// Tests for the command dispatch of BROTLib.FB_Comm_MQTT_Influx (BROTLib#39): single-field messages as pyBROT and
// BROTgui send them, and multi-field messages where track/slew must see the data of the same message. The handler is
// called directly with a payload; no MQTT connection is made. A stub records what it asks the telescope to do.
FUNCTION_BLOCK FB_Comm_MQTT_Influx_Tests EXTENDS TcUnit.FB_TestSuite
VAR
	fbComm	: BROTLib.FB_Comm_MQTT_Influx;
	stub	: FB_TelescopeStub;
	bReady	: BOOL;
	bSingle_Field_Messages_Still_Fill_The_Buffer	: BOOL;
	bData_Before_Verb_In_One_Message	: BOOL;
	bVerb_First_Uses_Data_From_The_Same_Message	: BOOL;
	bSame_Message_Data_Beats_The_Buffer	: BOOL;
	bIncomplete_Pair_Is_Dropped	: BOOL;
	bBuffer_Is_Cleared_After_Track	: BOOL;
	bSlew_Takes_Elevation_And_Azimuth_From_One_Message	: BOOL;
	bTrailing_Timestamp_Does_Not_Break_The_Last_Field	: BOOL;
	bOther_Measurement_Is_Ignored	: BOOL;
	bFields_Beyond_The_Eighth_Are_Ignored	: BOOL;
	bNon_Numeric_Coordinate_Is_Rejected	: BOOL;
	bOut_Of_Range_Coordinates_Are_Rejected	: BOOL;
	bRange_Limits_Are_Accepted	: BOOL;
	bRejected_Value_Clears_The_Buffer	: BOOL;
END_VAR

IF NOT bReady THEN
	bReady := TRUE;
	fbComm.Telescope := stub;
END_IF
Single_Field_Messages_Still_Fill_The_Buffer();
Data_Before_Verb_In_One_Message();
Verb_First_Uses_Data_From_The_Same_Message();
Same_Message_Data_Beats_The_Buffer();
Incomplete_Pair_Is_Dropped();
Buffer_Is_Cleared_After_Track();
Slew_Takes_Elevation_And_Azimuth_From_One_Message();
Trailing_Timestamp_Does_Not_Break_The_Last_Field();
Other_Measurement_Is_Ignored();
Fields_Beyond_The_Eighth_Are_Ignored();
Non_Numeric_Coordinate_Is_Rejected();
Out_Of_Range_Coordinates_Are_Rejected();
Range_Limits_Are_Accepted();
Rejected_Value_Clears_The_Buffer();

// Puts the handler and the stub back to a clean state; every test runs its body once.
METHOD PRIVATE ResetHandler
VAR_INPUT
END_VAR
// drain whatever the previous test left in the handler's buffers: track and slew consume and clear them
fbComm._handleMQTTMessage(sPayloadRcv := 'command track=1');
fbComm._handleMQTTMessage(sPayloadRcv := 'command slew=1');
stub.ClearCounters();
END_METHOD

// The way pyBROT and BROTgui send it today: three messages, the buffer is consumed by track.
METHOD PRIVATE Single_Field_Messages_Still_Fill_The_Buffer
VAR
END_VAR
TEST('Single_Field_Messages_Still_Fill_The_Buffer');
IF NOT bSingle_Field_Messages_Still_Fill_The_Buffer THEN
	bSingle_Field_Messages_Still_Fill_The_Buffer := TRUE;
	ResetHandler();
	fbComm._handleMQTTMessage(sPayloadRcv := 'command rightascension=10.5');
	fbComm._handleMQTTMessage(sPayloadRcv := 'command declination=20.5');
	AssertEquals_INT(Expected := 0, Actual := stub.nTrack, Message := 'before track: number of Track calls');
	fbComm._handleMQTTMessage(sPayloadRcv := 'command track=1');
	AssertEquals_INT(Expected := 1, Actual := stub.nTrack, Message := 'after track: number of Track calls');
	AssertEquals_LREAL(Expected := 10.5, Actual := stub.fTrackRa, Delta := 1.0E-9, Message := 'after track: right ascension');
	AssertEquals_LREAL(Expected := 20.5, Actual := stub.fTrackDec, Delta := 1.0E-9, Message := 'after track: declination');
	TEST_FINISHED();
END_IF
END_METHOD

METHOD PRIVATE Data_Before_Verb_In_One_Message
VAR
END_VAR
TEST('Data_Before_Verb_In_One_Message');
IF NOT bData_Before_Verb_In_One_Message THEN
	bData_Before_Verb_In_One_Message := TRUE;
	ResetHandler();
	fbComm._handleMQTTMessage(sPayloadRcv := 'command rightascension=10.5,declination=20.5,track=1');
	AssertEquals_INT(Expected := 1, Actual := stub.nTrack, Message := 'one message: number of Track calls');
	AssertEquals_LREAL(Expected := 10.5, Actual := stub.fTrackRa, Delta := 1.0E-9, Message := 'one message: right ascension');
	AssertEquals_LREAL(Expected := 20.5, Actual := stub.fTrackDec, Delta := 1.0E-9, Message := 'one message: declination');
	TEST_FINISHED();
END_IF
END_METHOD

// The data pass runs before the verb pass, so the field order does not matter.
METHOD PRIVATE Verb_First_Uses_Data_From_The_Same_Message
VAR
END_VAR
TEST('Verb_First_Uses_Data_From_The_Same_Message');
IF NOT bVerb_First_Uses_Data_From_The_Same_Message THEN
	bVerb_First_Uses_Data_From_The_Same_Message := TRUE;
	ResetHandler();
	fbComm._handleMQTTMessage(sPayloadRcv := 'command track=1,rightascension=10.5,declination=20.5');
	AssertEquals_INT(Expected := 1, Actual := stub.nTrack, Message := 'verb first: number of Track calls');
	AssertEquals_LREAL(Expected := 10.5, Actual := stub.fTrackRa, Delta := 1.0E-9, Message := 'verb first: right ascension');
	AssertEquals_LREAL(Expected := 20.5, Actual := stub.fTrackDec, Delta := 1.0E-9, Message := 'verb first: declination');
	TEST_FINISHED();
END_IF
END_METHOD

// An old buffer value must never be combined with the new target.
METHOD PRIVATE Same_Message_Data_Beats_The_Buffer
VAR
END_VAR
TEST('Same_Message_Data_Beats_The_Buffer');
IF NOT bSame_Message_Data_Beats_The_Buffer THEN
	bSame_Message_Data_Beats_The_Buffer := TRUE;
	ResetHandler();
	fbComm._handleMQTTMessage(sPayloadRcv := 'command rightascension=1.5');
	fbComm._handleMQTTMessage(sPayloadRcv := 'command declination=2.5');
	fbComm._handleMQTTMessage(sPayloadRcv := 'command rightascension=10.5,declination=20.5,track=1');
	AssertEquals_INT(Expected := 1, Actual := stub.nTrack, Message := 'stale buffer: number of Track calls');
	AssertEquals_LREAL(Expected := 10.5, Actual := stub.fTrackRa, Delta := 1.0E-9, Message := 'stale buffer: right ascension');
	AssertEquals_LREAL(Expected := 20.5, Actual := stub.fTrackDec, Delta := 1.0E-9, Message := 'stale buffer: declination');
	TEST_FINISHED();
END_IF
END_METHOD

// Same as the buffered form: no declination, no Track call.
METHOD PRIVATE Incomplete_Pair_Is_Dropped
VAR
END_VAR
TEST('Incomplete_Pair_Is_Dropped');
IF NOT bIncomplete_Pair_Is_Dropped THEN
	bIncomplete_Pair_Is_Dropped := TRUE;
	ResetHandler();
	fbComm._handleMQTTMessage(sPayloadRcv := 'command rightascension=10.5,track=1');
	AssertEquals_INT(Expected := 0, Actual := stub.nTrack, Message := 'declination missing: number of Track calls');
	TEST_FINISHED();
END_IF
END_METHOD

// The second track finds an empty buffer and is dropped, the first call stays the last one.
METHOD PRIVATE Buffer_Is_Cleared_After_Track
VAR
END_VAR
TEST('Buffer_Is_Cleared_After_Track');
IF NOT bBuffer_Is_Cleared_After_Track THEN
	bBuffer_Is_Cleared_After_Track := TRUE;
	ResetHandler();
	fbComm._handleMQTTMessage(sPayloadRcv := 'command rightascension=10.5,declination=20.5,track=1');
	fbComm._handleMQTTMessage(sPayloadRcv := 'command track=1');
	AssertEquals_INT(Expected := 1, Actual := stub.nTrack, Message := 'second track without data: number of Track calls');
	AssertEquals_LREAL(Expected := 10.5, Actual := stub.fTrackRa, Delta := 1.0E-9, Message := 'second track without data: right ascension');
	AssertEquals_LREAL(Expected := 20.5, Actual := stub.fTrackDec, Delta := 1.0E-9, Message := 'second track without data: declination');
	TEST_FINISHED();
END_IF
END_METHOD

METHOD PRIVATE Slew_Takes_Elevation_And_Azimuth_From_One_Message
VAR
END_VAR
TEST('Slew_Takes_Elevation_And_Azimuth_From_One_Message');
IF NOT bSlew_Takes_Elevation_And_Azimuth_From_One_Message THEN
	bSlew_Takes_Elevation_And_Azimuth_From_One_Message := TRUE;
	ResetHandler();
	fbComm._handleMQTTMessage(sPayloadRcv := 'command slew=1,azimuth=120.5,elevation=45.5');
	AssertEquals_INT(Expected := 1, Actual := stub.nSlew, Message := 'slew: number of Slew calls');
	AssertEquals_LREAL(Expected := 120.5, Actual := stub.fSlewAz, Delta := 1.0E-9, Message := 'slew: azimuth');
	AssertEquals_LREAL(Expected := 45.5, Actual := stub.fSlewAlt, Delta := 1.0E-9, Message := 'slew: altitude');
	TEST_FINISHED();
END_IF
END_METHOD

METHOD PRIVATE Trailing_Timestamp_Does_Not_Break_The_Last_Field
VAR
END_VAR
TEST('Trailing_Timestamp_Does_Not_Break_The_Last_Field');
IF NOT bTrailing_Timestamp_Does_Not_Break_The_Last_Field THEN
	bTrailing_Timestamp_Does_Not_Break_The_Last_Field := TRUE;
	ResetHandler();
	fbComm._handleMQTTMessage(sPayloadRcv := 'command rightascension=10.5,declination=20.5,track=1 1700000000000000000');
	AssertEquals_INT(Expected := 1, Actual := stub.nTrack, Message := 'timestamp: number of Track calls');
	AssertEquals_LREAL(Expected := 10.5, Actual := stub.fTrackRa, Delta := 1.0E-9, Message := 'timestamp: right ascension');
	AssertEquals_LREAL(Expected := 20.5, Actual := stub.fTrackDec, Delta := 1.0E-9, Message := 'timestamp: declination');
	TEST_FINISHED();
END_IF
END_METHOD

METHOD PRIVATE Other_Measurement_Is_Ignored
VAR
END_VAR
TEST('Other_Measurement_Is_Ignored');
IF NOT bOther_Measurement_Is_Ignored THEN
	bOther_Measurement_Is_Ignored := TRUE;
	ResetHandler();
	fbComm._handleMQTTMessage(sPayloadRcv := 'status rightascension=10.5,declination=20.5,track=1');
	AssertEquals_INT(Expected := 0, Actual := stub.nTrack, Message := 'measurement status: number of Track calls');
	TEST_FINISHED();
END_IF
END_METHOD

// At most 8 fields per message (a malformed message must not spin the scan cycle); the rest is logged and ignored.
METHOD PRIVATE Fields_Beyond_The_Eighth_Are_Ignored
VAR
END_VAR
TEST('Fields_Beyond_The_Eighth_Are_Ignored');
IF NOT bFields_Beyond_The_Eighth_Are_Ignored THEN
	bFields_Beyond_The_Eighth_Are_Ignored := TRUE;
	ResetHandler();
	fbComm._handleMQTTMessage(sPayloadRcv := 'command rightascension=10.5,declination=20.5,x1=0,x2=0,x3=0,x4=0,x5=0,x6=0,track=1');
	AssertEquals_INT(Expected := 0, Actual := stub.nTrack, Message := 'track is the ninth field: number of Track calls');
	TEST_FINISHED();
END_IF
END_METHOD

// STRING_TO_LREAL turns garbage into 0.0, a valid coordinate; it must not reach Track (#27).
METHOD PRIVATE Non_Numeric_Coordinate_Is_Rejected
VAR
END_VAR
TEST('Non_Numeric_Coordinate_Is_Rejected');
IF NOT bNon_Numeric_Coordinate_Is_Rejected THEN
	bNon_Numeric_Coordinate_Is_Rejected := TRUE;
	ResetHandler();
	fbComm._handleMQTTMessage(sPayloadRcv := 'command rightascension=abc,declination=20.5,track=1');
	AssertEquals_INT(Expected := 0, Actual := stub.nTrack, Message := 'rightascension=abc: number of Track calls');
	fbComm._handleMQTTMessage(sPayloadRcv := 'command rightascension=10.5,declination=nan,track=1');
	AssertEquals_INT(Expected := 0, Actual := stub.nTrack, Message := 'declination=nan: number of Track calls');
	TEST_FINISHED();
END_IF
END_METHOD

METHOD PRIVATE Out_Of_Range_Coordinates_Are_Rejected
VAR
END_VAR
TEST('Out_Of_Range_Coordinates_Are_Rejected');
IF NOT bOut_Of_Range_Coordinates_Are_Rejected THEN
	bOut_Of_Range_Coordinates_Are_Rejected := TRUE;
	ResetHandler();
	fbComm._handleMQTTMessage(sPayloadRcv := 'command rightascension=10.5,declination=95,track=1');
	AssertEquals_INT(Expected := 0, Actual := stub.nTrack, Message := 'declination=95: number of Track calls');
	fbComm._handleMQTTMessage(sPayloadRcv := 'command rightascension=1e999,declination=20.5,track=1');
	AssertEquals_INT(Expected := 0, Actual := stub.nTrack, Message := 'rightascension=1e999: number of Track calls');
	fbComm._handleMQTTMessage(sPayloadRcv := 'command elevation=120,azimuth=10,slew=1');
	AssertEquals_INT(Expected := 0, Actual := stub.nSlew, Message := 'elevation=120: number of Slew calls');
	TEST_FINISHED();
END_IF
END_METHOD

// The limits themselves are valid values; so are signs and exponents.
METHOD PRIVATE Range_Limits_Are_Accepted
VAR
END_VAR
TEST('Range_Limits_Are_Accepted');
IF NOT bRange_Limits_Are_Accepted THEN
	bRange_Limits_Are_Accepted := TRUE;
	ResetHandler();
	fbComm._handleMQTTMessage(sPayloadRcv := 'command rightascension=0,declination=-90,track=1');
	AssertEquals_INT(Expected := 1, Actual := stub.nTrack, Message := 'ra=0, dec=-90: number of Track calls');
	fbComm._handleMQTTMessage(sPayloadRcv := 'command rightascension=360,declination=+9e1,track=1');
	AssertEquals_INT(Expected := 2, Actual := stub.nTrack, Message := 'ra=360, dec=+9e1: number of Track calls');
	AssertEquals_LREAL(Expected := 90.0, Actual := stub.fTrackDec, Delta := 1.0E-9, Message := 'dec=+9e1: declination');
	TEST_FINISHED();
END_IF
END_METHOD

// A rejected coordinate must not fall back to one buffered by an earlier message: the track is dropped instead.
METHOD PRIVATE Rejected_Value_Clears_The_Buffer
VAR
END_VAR
TEST('Rejected_Value_Clears_The_Buffer');
IF NOT bRejected_Value_Clears_The_Buffer THEN
	bRejected_Value_Clears_The_Buffer := TRUE;
	ResetHandler();
	fbComm._handleMQTTMessage(sPayloadRcv := 'command rightascension=1.5');
	fbComm._handleMQTTMessage(sPayloadRcv := 'command rightascension=abc,declination=20.5,track=1');
	AssertEquals_INT(Expected := 0, Actual := stub.nTrack, Message := 'buffered ra, then ra=abc: number of Track calls');
	TEST_FINISHED();
END_IF
END_METHOD

END_FUNCTION_BLOCK

(* stored: Version 1.1.0.1, ProductVersion 3.1.4024.15
   POU FB_Comm_MQTT_Influx_Tests: Id {34557123-6b20-450c-8e1e-e569b4e30879}, SpecialFunc None
   Method ResetHandler: Id {e4163f5e-60d4-4240-b519-3bcc1b5eb9d9}
   Method Single_Field_Messages_Still_Fill_The_Buffer: Id {bf448ccc-63d8-435d-9991-76e2552690de}
   Method Data_Before_Verb_In_One_Message: Id {3a11763f-f81c-4a99-9829-5ab118ed367b}
   Method Verb_First_Uses_Data_From_The_Same_Message: Id {e8a94e9c-48f1-4ccd-a98c-22d7e10d0a9a}
   Method Same_Message_Data_Beats_The_Buffer: Id {a02743b4-6532-4b68-8837-639d84cd727f}
   Method Incomplete_Pair_Is_Dropped: Id {fd35e970-9a15-4f5c-98a3-32b668e2db14}
   Method Buffer_Is_Cleared_After_Track: Id {72b7c574-480d-4146-8423-48463225227c}
   Method Slew_Takes_Elevation_And_Azimuth_From_One_Message: Id {ed1e6218-9e8f-429c-99e1-f69d844d24e7}
   Method Trailing_Timestamp_Does_Not_Break_The_Last_Field: Id {7eed211b-d43a-4fa7-ba14-ab60aba02482}
   Method Other_Measurement_Is_Ignored: Id {7311dfe5-1b87-4e83-b0cf-0c4bd649d7e3}
   Method Fields_Beyond_The_Eighth_Are_Ignored: Id {e6b89235-1e3d-47b1-8a05-9b4fa04bbd63}
   Method Non_Numeric_Coordinate_Is_Rejected: Id {70e0277b-64c7-4892-988c-3be963d7f592}
   Method Out_Of_Range_Coordinates_Are_Rejected: Id {c629a73e-2263-4856-a25c-456cd6c5bfe9}
   Method Range_Limits_Are_Accepted: Id {2234caa2-2a82-426e-91ed-05b02e9efd06}
   Method Rejected_Value_Clears_The_Buffer: Id {70e7ff01-12c5-4d27-8596-129dcb4f5565} *)
